{attribute 'Tc2GvlVarNames'}
{attribute 'strict'}
TYPE e_ProgrammiMovimentoX :
(
	
	X_PosDiRiposo					:= 0,
	X_PosFuoriIngombroRiposo 			:= 6,

	X_PosPrelievoFalda					:= 51,
	X_PosDepositoSuCatastaFalda			:= 52,
	X_PosDepositoFalda					:= 53,
	X_PosFuoriIngombroVuotoFalda		:= 56,

	X_PosStartLentaPrelievoLastra 		:= 101,
	X_PosPrelievoInLentaLastra 			:= 102,
	X_PosDistaccoLastraInLentaLastra	:= 103,
	X_PosStartLentaDepositoLastra 		:= 104,
	X_PosDepositoInLentaLastra			:= 105,
	X_PosFuoriIngombroVuotoLastra		:= 106,
	X_PosFuoriIngombroCaricoLastra		:= 126,
	X_PosGiroPiezaTraCavallete			:= 127
);
END_TYPE

(* stored: Version 1.1.0.1, ProductVersion 3.1.4024.11
   EnumerationTextList e_ProgrammiMovimentoX: Id {d322e122-b2d0-4221-ae96-2ed60d8a721f} *)
